TYPE ST_LeakTester_CycleData :
STRUCT

	aLeakTesterLastResult			: st_i28LasResult;

END_STRUCT
END_TYPE

(* stored: Version 1.1.0.1, ProductVersion 3.1.4024.13
   DUT ST_LeakTester_CycleData: Id {a87f5642-6635-4d10-aef6-f9a75b94d380} *)
